FUNCTION_BLOCK RunUnitGeneric Extends CommonBase
VAR_INPUT
	bEnStep : BOOL;
	bTrigStep : BOOL;
	bPause : BOOL;
	bIsBypassed : BOOL;
	bWorkingOverride : BOOL;
	bMaterialOverride : BOOL;
	
	slaveWorkingSignal : ARRAY[1..32] OF BOOL; // collect slave working signal , possible to access externally?
END_VAR
VAR_OUTPUT
	State : INT := 0;
	NextState : INT := 0;
	AlarmCode : UDINT := 0;
END_VAR
VAR	
	Parent : POINTER TO RunUnitGeneric;
	
	SlotBase : POINTER TO MaterialBlock;
	SlotCount : int ;
	SlotLast : POINTER TO MaterialBlock;
	
	bLastParentStatus : BIT; // memorize last parent status	
	bSerialTransition : BIT;
	transitionByte : BYTE;
	
	isTransit : BOOL ;
	workingTimer : LTON;
	
	outputState : int;
END_VAR
VAR PERSISTENT
	//station specific settings area (user settings
	slaveLinkageStatus : ARRAY[1..32] OF BOOL; // configuration
	miscsParameters : ARRAY[1..8] of int;
END_VAR
VAR CONSTANT 
	bit0EnStep : INT := 0;
	bit1TrigStep : INT := 1;
	bit2StatePause : INT :=2;
	bit3IsBypassed : INT :=3;
	bit4WorkingOverride : INT :=4;
	bit5MaterialOverride : INT :=5;
END_VAR


//Catch parent's pause status
IF Parent^.bPause AND NOT bLastParentStatus THEN
	bPause := TRUE;
END_IF

IF NOT Parent^.bPause AND bPause THEN
	bPause := FALSE;
END_IF

bLastParentStatus := Parent^.bPause;

//Serial transition
IF bSerialTransition AND (State = NextState) THEN
	NextState := State +1 ;
END_IF

//Reset transition word
IF NextState <> State THEN
	transitionByte := 0;
	bSerialTransition := FALSE;
	AlarmCode := 0;
	
	State := NextState; //release and go
END_IF


//transit condition
isTransit := (NOT bEnStep OR (bEnStep AND bTrigStep)) AND NOT bPause;

IF isTransit THEN
	outputState := State; //release and go
ELSE
	outputState := eSpecialStates.FORBIDDEN;
END_IF

//Reset trigger step
bTrigStep := FALSE;

//Timer
workingTimer(IN:=,PT:=,Q=>,ET=>);

METHOD ConfigureRead : CellDataBlock
VAR_INPUT
	mode : eModes;
END_VAR
END_METHOD

METHOD ConfigureWrite : BOOL
VAR_INPUT
	input : CellDataBlock;
	mode : eModes;
END_VAR
//Implemented by concre derived class
END_METHOD

METHOD Control : BOOL
VAR_INPUT
	input : CellDataBlock;
	mode : eModes; //commit mode
END_VAR
bEnStep := input.unit.base.controlWord.bit0EnStep;
bTrigStep := input.unit.base.controlWord.bit1TrigStep;
bPause := input.unit.base.controlWord.bit2StatePause;
bIsBypassed := input.unit.base.controlWord.bit3IsBypassed;
bWorkingOverride := input.unit.base.controlWord.bit4WorkingOverride;
bMaterialOverride := input.unit.base.controlWord.bit5MaterialOverride;
Control:=true;
END_METHOD

METHOD ErrorClear : BOOL
VAR_INPUT
	input : eErrorClearWays;
END_VAR
AlarmCode := 0; //code reset to 0
END_METHOD

METHOD ErrorDetect : UDINT
VAR_INPUT
END_VAR
ErrorDetect := AlarmCode;
END_METHOD

METHOD FB_init : BOOL
VAR_INPUT
	bInitRetains : BOOL; // if TRUE, the retain variables are initialized (warm start / cold start)
	bInCopyCode : BOOL;  // if TRUE, the instance afterwards gets moved into the copy code (online change)
	
	argParent : POINTER TO RunUnitGeneric;
	argSlotBase : POINTER TO MaterialBlock;
	argSlotLast : POINTER TO MaterialBlock;
END_VAR
//initialize 
Parent := argParent;
SlotBase := argSlotBase;
SlotLast := argSlotLast;
//
IF bInitRetains THEN
	NextState := eSpecialStates.INITIAL_BEGIN;
END_IF
END_METHOD

METHOD Initialize : BOOL
VAR_INPUT
END_VAR
//once initializing method call , redirect current state to initalizing region
IF (TO_UINT(State) AND TO_UINT(eSpecialStates.INITIAL_REGION)) =0 THEN
	NextState := eSpecialStates.INITIAL_BEGIN; //not in intializing region , change
END_IF

Initialize := (State = eSpecialStates.INITIAL_END);
END_METHOD

METHOD Monitor : CellDataBlock
VAR_INPUT
END_VAR
Monitor.unit.base.controlWord.bit0EnStep := bEnStep;
Monitor.unit.base.controlWord.bit1TrigStep := bTrigStep;
Monitor.unit.base.controlWord.bit2StatePause := bPause;
Monitor.unit.base.controlWord.bit3IsBypassed := bIsBypassed;
Monitor.unit.base.controlWord.bit4WorkingOverride := bWorkingOverride;
Monitor.unit.base.controlWord.bit5MaterialOverride := bMaterialOverride;
//Transition status
Monitor.unit.base.transitionByte := transitionByte;
//
Monitor.unit.base.alarmCode := TO_WORD(AlarmCode);
Monitor.unit.base.state := TO_WORD(State);
Monitor.unit.base.nextState := TO_WORD(NextState);
//
Monitor.unit.base.workingTimerCache := TO_DWORD(workingTimer.ET);
END_METHOD

METHOD TypeCode : eCategrories
VAR_INPUT
END_VAR
TypeCode := eCategrories.SELECTION_UNIT;
END_METHOD

END_FUNCTION_BLOCK

(* stored: Version 1.1.0.1, ProductVersion 3.1.4022.10
   POU RunUnitGeneric: Id {a108e392-1419-4492-a6fc-c3186312016b}, SpecialFunc None
   Folder CommonBase: Id {a3eb2459-fb17-4657-a789-38e4b978c786}
   Method ConfigureRead: Id {5b0d9a0a-5d92-42f2-80d6-58161cf4acad}
   Method ConfigureWrite: Id {b15520cc-2020-48bd-8025-beb0523946ca}
   Method Control: Id {fe69a240-a6bf-45a3-bd63-78ff17e8577a}
   Method ErrorClear: Id {c0e62209-d0d5-44f2-8c68-278b3588f780}
   Method ErrorDetect: Id {f4463e33-7efc-4b67-a80e-02e00ed76350}
   Method FB_init: Id {1054404a-900b-4aa2-9841-9d1387599ab2}
   Method Initialize: Id {54b8cb88-45e4-469a-a3ac-c4ff2e84617d}
   Method Monitor: Id {8df8139c-9882-4bf6-9048-c2ce81b63c35}
   Method TypeCode: Id {5f35ce6c-c451-4e46-809f-fa5a3eec0aed} *)
